// Mitsubishi GX Works2 project: LRI - PLC - SELO   PLC: Q03UDV

PROGRAM MAIN
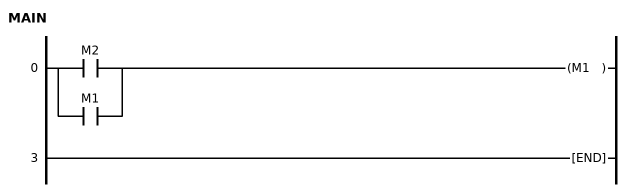
0     LD      M2
      OR      M1
      OUT     M1
3     END
END_PROGRAM
